// TIA Portal project "SuperSygnalizacjaDomiLechLuka" (V16)

(* hardware
DEVICE "S7-1200 station_2"  S7-1200 Station
   slot 0: "Rack_0"  S7-1200 Rack  Rack  V1.0
   slot 1: "PLC_2"  CPU 1215C AC/DC/Rly  6ES7 215-1BG40-0XB0  V4.4
DEVICE "S7-1200 station_1"  S7-1200 Station
   slot 0: "Rack_0"  S7-1200 Rack  Rack  V1.0
   slot 1: "PLC_1"  CPU 1215C AC/DC/Rly  6ES7 215-1BG40-0XB0  V4.4
*)

// ===== PLC "PLC_1"  CPU 1215C AC/DC/Rly =====

VAR_GLOBAL   // PLC tag table "Default tag table"
   "Clock_Byte" AT %MB0 : Byte;
   "Clock_10Hz" AT %M0.0 : Bool;
   "Clock_5Hz" AT %M0.1 : Bool;
   "Clock_2.5Hz" AT %M0.2 : Bool;
   "Clock_2Hz" AT %M0.3 : Bool;
   "Clock_1.25Hz" AT %M0.4 : Bool;
   "Clock_1Hz" AT %M0.5 : Bool;
   "Clock_0.625Hz" AT %M0.6 : Bool;
   "Clock_0.5Hz" AT %M0.7 : Bool;
   "P3_P4_green" AT %Q0.0 : Bool;
   "P3_P4_red" AT %Q0.1 : Bool;
   "W1_W3_W4_red" AT %Q0.2 : Bool;
   "W1_W3_W4_yellow" AT %Q0.3 : Bool;
   "W1_W3_W4_green" AT %Q0.4 : Bool;
   "W2_W6_red" AT %Q0.5 : Bool;
   "W2_W6_yellow" AT %Q0.6 : Bool;
   "W2_W6_green" AT %Q0.7 : Bool;
   "P2_red" AT %Q1.0 : Bool;
   "Start" AT %M1.0 : Bool;
   "Timer_CV" AT %MD10 : DWord;
   "P2_green" AT %M1.1 : Bool;
   "W7_red" AT %M1.2 : Bool;
   "W7_yellow" AT %M1.3 : Bool;
   "W7_green" AT %M1.4 : Bool;
   "W5_red" AT %M1.5 : Bool;
   "W5_yellow" AT %M1.6 : Bool;
   "W5_green" AT %M1.7 : Bool;
   "P1_red" AT %M2.0 : Bool;
   "P1_green" AT %M2.1 : Bool;
END_VAR

DATA_BLOCK "sent"   // DB1
{ S7_Optimized_Access := 'TRUE' }
VERSION : 0.1
   VAR
      data : Word;
   END_VAR
BEGIN
END_DATA_BLOCK

DATA_BLOCK "recv"   // DB2
{ S7_Optimized_Access := 'TRUE' }
VERSION : 0.1
   VAR
      data : Word;
   END_VAR
BEGIN
END_DATA_BLOCK

// folder: System blocks/Program resources

DATA_BLOCK "IEC_Timer_0_DB"   // DB3
{ S7_Optimized_Access := 'TRUE' }
AUTHOR : Simatic
FAMILY : IEC
NAME : IEC_TMR
VERSION : 1.0
// stored: InstanceOfName IEC_TIMER
"IEC_TIMER"
BEGIN
END_DATA_BLOCK

// folder: (top level)

ORGANIZATION_BLOCK "Main"   // OB1, LAD, ProgramCycle
TITLE = "Main Program Sweep (Cycle)"
{ S7_Optimized_Access := 'TRUE' }
VERSION : 0.1
   VAR_INPUT
      Initial_Call : Bool;   // Initial call of this OB
      Remanence : Bool;   // =True, if remanent data are available
   END_VAR
BEGIN

REGION Network 1: Main timer
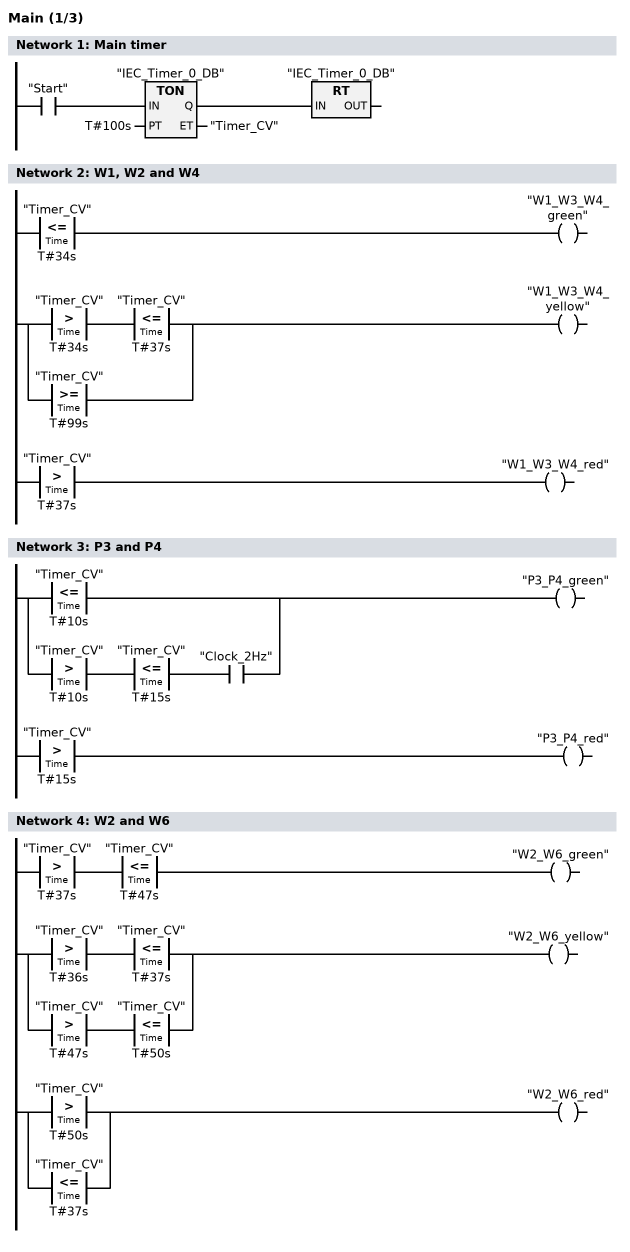
   "IEC_Timer_0_DB".TON(IN := "Start", PT := T#100s, ET => "Timer_CV");
   IF "IEC_Timer_0_DB".Q THEN RESET_TIMER("IEC_Timer_0_DB"); END_IF;
END_REGION

REGION Network 2: W1, W2 and W4
   RUNG wire#powerrail
      { S7_Templates := "SrcType := Time" } LE_Contact(in1 := "Timer_CV", in2 := T#34s)
      Coil( "W1_W3_W4_green" )
   END_RUNG
   RUNG wire#powerrail
      { S7_Templates := "SrcType := Time" } GT_Contact(in1 := "Timer_CV", in2 := T#34s)
      { S7_Templates := "SrcType := Time" } LE_Contact(in1 := "Timer_CV", in2 := T#37s)
      wire#w1
      Coil( "W1_W3_W4_yellow" )
   END_RUNG
   RUNG wire#powerrail
      { S7_Templates := "SrcType := Time" } GE_Contact(in1 := "Timer_CV", in2 := T#99s)
   END_RUNG wire#w1
   RUNG wire#powerrail
      { S7_Templates := "SrcType := Time" } GT_Contact(in1 := "Timer_CV", in2 := T#37s)
      Coil( "W1_W3_W4_red" )
   END_RUNG
   // the same network as SCL:
   "W1_W3_W4_green" := "Timer_CV" <= T#34s;
   "W1_W3_W4_yellow" := (("Timer_CV" > T#34s) AND ("Timer_CV" <= T#37s)) OR ("Timer_CV" >= T#99s);
   "W1_W3_W4_red" := "Timer_CV" > T#37s;
END_REGION

REGION Network 3: P3 and P4
   RUNG wire#powerrail
      { S7_Templates := "SrcType := Time" } LE_Contact(in1 := "Timer_CV", in2 := T#10s)
      wire#w1
      Coil( "P3_P4_green" )
   END_RUNG
   RUNG wire#powerrail
      { S7_Templates := "SrcType := Time" } GT_Contact(in1 := "Timer_CV", in2 := T#10s)
      { S7_Templates := "SrcType := Time" } LE_Contact(in1 := "Timer_CV", in2 := T#15s)
      Contact( "Clock_2Hz" )
   END_RUNG wire#w1
   RUNG wire#powerrail
      { S7_Templates := "SrcType := Time" } GT_Contact(in1 := "Timer_CV", in2 := T#15s)
      Coil( "P3_P4_red" )
   END_RUNG
   // the same network as SCL:
   "P3_P4_green" := ("Timer_CV" <= T#10s) OR (("Timer_CV" > T#10s) AND ("Timer_CV" <= T#15s) AND "Clock_2Hz");
   "P3_P4_red" := "Timer_CV" > T#15s;
END_REGION

REGION Network 4: W2 and W6
   RUNG wire#powerrail
      { S7_Templates := "SrcType := Time" } GT_Contact(in1 := "Timer_CV", in2 := T#37s)
      { S7_Templates := "SrcType := Time" } LE_Contact(in1 := "Timer_CV", in2 := T#47s)
      Coil( "W2_W6_green" )
   END_RUNG
   RUNG wire#powerrail
      { S7_Templates := "SrcType := Time" } GT_Contact(in1 := "Timer_CV", in2 := T#36s)
      { S7_Templates := "SrcType := Time" } LE_Contact(in1 := "Timer_CV", in2 := T#37s)
      wire#w1
      Coil( "W2_W6_yellow" )
   END_RUNG
   RUNG wire#powerrail
      { S7_Templates := "SrcType := Time" } GT_Contact(in1 := "Timer_CV", in2 := T#47s)
      { S7_Templates := "SrcType := Time" } LE_Contact(in1 := "Timer_CV", in2 := T#50s)
   END_RUNG wire#w1
   RUNG wire#powerrail
      { S7_Templates := "SrcType := Time" } GT_Contact(in1 := "Timer_CV", in2 := T#50s)
      wire#w2
      Coil( "W2_W6_red" )
   END_RUNG
   RUNG wire#powerrail
      { S7_Templates := "SrcType := Time" } LE_Contact(in1 := "Timer_CV", in2 := T#37s)
   END_RUNG wire#w2
   // the same network as SCL:
   "W2_W6_green" := ("Timer_CV" > T#37s) AND ("Timer_CV" <= T#47s);
   "W2_W6_yellow" := (("Timer_CV" > T#36s) AND ("Timer_CV" <= T#37s)) OR (("Timer_CV" > T#47s) AND ("Timer_CV" <= T#50s));
   "W2_W6_red" := ("Timer_CV" > T#50s) OR ("Timer_CV" <= T#37s);
END_REGION

REGION Network 5: P2
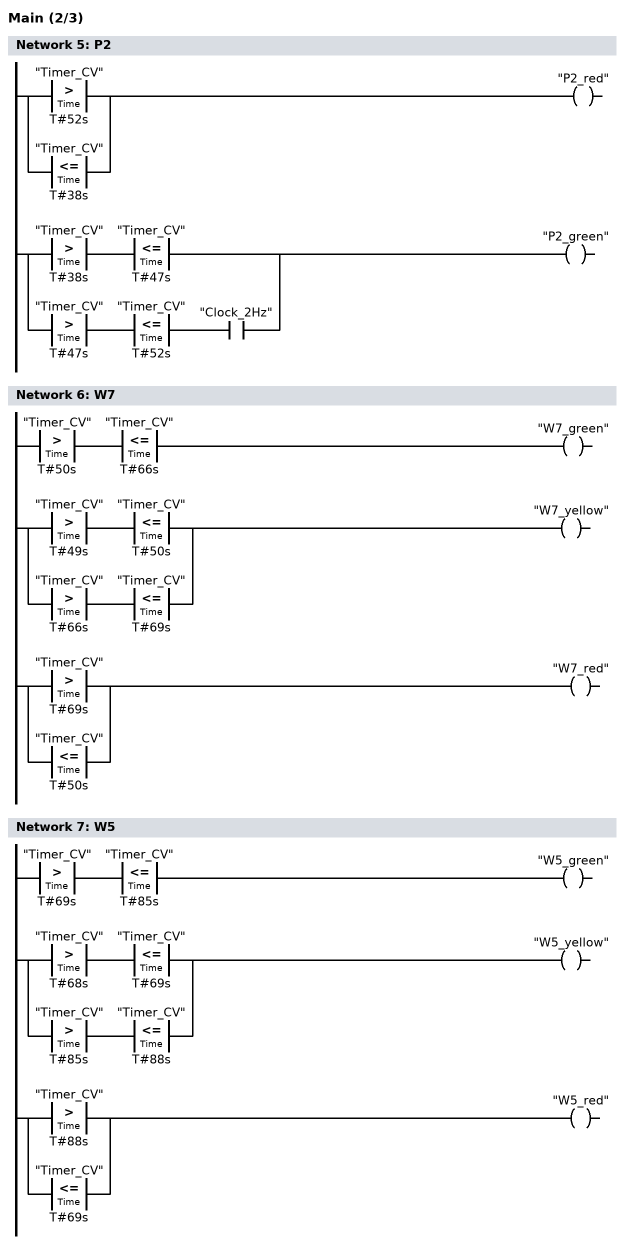
   RUNG wire#powerrail
      { S7_Templates := "SrcType := Time" } GT_Contact(in1 := "Timer_CV", in2 := T#52s)
      wire#w1
      Coil( "P2_red" )
   END_RUNG
   RUNG wire#powerrail
      { S7_Templates := "SrcType := Time" } LE_Contact(in1 := "Timer_CV", in2 := T#38s)
   END_RUNG wire#w1
   RUNG wire#powerrail
      { S7_Templates := "SrcType := Time" } GT_Contact(in1 := "Timer_CV", in2 := T#38s)
      { S7_Templates := "SrcType := Time" } LE_Contact(in1 := "Timer_CV", in2 := T#47s)
      wire#w2
      Coil( "P2_green" )
   END_RUNG
   RUNG wire#powerrail
      { S7_Templates := "SrcType := Time" } GT_Contact(in1 := "Timer_CV", in2 := T#47s)
      { S7_Templates := "SrcType := Time" } LE_Contact(in1 := "Timer_CV", in2 := T#52s)
      Contact( "Clock_2Hz" )
   END_RUNG wire#w2
   // the same network as SCL:
   "P2_red" := ("Timer_CV" > T#52s) OR ("Timer_CV" <= T#38s);
   "P2_green" := (("Timer_CV" > T#38s) AND ("Timer_CV" <= T#47s)) OR (("Timer_CV" > T#47s) AND ("Timer_CV" <= T#52s) AND "Clock_2Hz");
END_REGION

REGION Network 6: W7
   RUNG wire#powerrail
      { S7_Templates := "SrcType := Time" } GT_Contact(in1 := "Timer_CV", in2 := T#50s)
      { S7_Templates := "SrcType := Time" } LE_Contact(in1 := "Timer_CV", in2 := T#66s)
      Coil( "W7_green" )
   END_RUNG
   RUNG wire#powerrail
      { S7_Templates := "SrcType := Time" } GT_Contact(in1 := "Timer_CV", in2 := T#49s)
      { S7_Templates := "SrcType := Time" } LE_Contact(in1 := "Timer_CV", in2 := T#50s)
      wire#w1
      Coil( "W7_yellow" )
   END_RUNG
   RUNG wire#powerrail
      { S7_Templates := "SrcType := Time" } GT_Contact(in1 := "Timer_CV", in2 := T#66s)
      { S7_Templates := "SrcType := Time" } LE_Contact(in1 := "Timer_CV", in2 := T#69s)
   END_RUNG wire#w1
   RUNG wire#powerrail
      { S7_Templates := "SrcType := Time" } GT_Contact(in1 := "Timer_CV", in2 := T#69s)
      wire#w2
      Coil( "W7_red" )
   END_RUNG
   RUNG wire#powerrail
      { S7_Templates := "SrcType := Time" } LE_Contact(in1 := "Timer_CV", in2 := T#50s)
   END_RUNG wire#w2
   // the same network as SCL:
   "W7_green" := ("Timer_CV" > T#50s) AND ("Timer_CV" <= T#66s);
   "W7_yellow" := (("Timer_CV" > T#49s) AND ("Timer_CV" <= T#50s)) OR (("Timer_CV" > T#66s) AND ("Timer_CV" <= T#69s));
   "W7_red" := ("Timer_CV" > T#69s) OR ("Timer_CV" <= T#50s);
END_REGION

REGION Network 7: W5
   RUNG wire#powerrail
      { S7_Templates := "SrcType := Time" } GT_Contact(in1 := "Timer_CV", in2 := T#69s)
      { S7_Templates := "SrcType := Time" } LE_Contact(in1 := "Timer_CV", in2 := T#85s)
      Coil( "W5_green" )
   END_RUNG
   RUNG wire#powerrail
      { S7_Templates := "SrcType := Time" } GT_Contact(in1 := "Timer_CV", in2 := T#68s)
      { S7_Templates := "SrcType := Time" } LE_Contact(in1 := "Timer_CV", in2 := T#69s)
      wire#w1
      Coil( "W5_yellow" )
   END_RUNG
   RUNG wire#powerrail
      { S7_Templates := "SrcType := Time" } GT_Contact(in1 := "Timer_CV", in2 := T#85s)
      { S7_Templates := "SrcType := Time" } LE_Contact(in1 := "Timer_CV", in2 := T#88s)
   END_RUNG wire#w1
   RUNG wire#powerrail
      { S7_Templates := "SrcType := Time" } GT_Contact(in1 := "Timer_CV", in2 := T#88s)
      wire#w2
      Coil( "W5_red" )
   END_RUNG
   RUNG wire#powerrail
      { S7_Templates := "SrcType := Time" } LE_Contact(in1 := "Timer_CV", in2 := T#69s)
   END_RUNG wire#w2
   // the same network as SCL:
   "W5_green" := ("Timer_CV" > T#69s) AND ("Timer_CV" <= T#85s);
   "W5_yellow" := (("Timer_CV" > T#68s) AND ("Timer_CV" <= T#69s)) OR (("Timer_CV" > T#85s) AND ("Timer_CV" <= T#88s));
   "W5_red" := ("Timer_CV" > T#88s) OR ("Timer_CV" <= T#69s);
END_REGION

REGION Network 8: P1
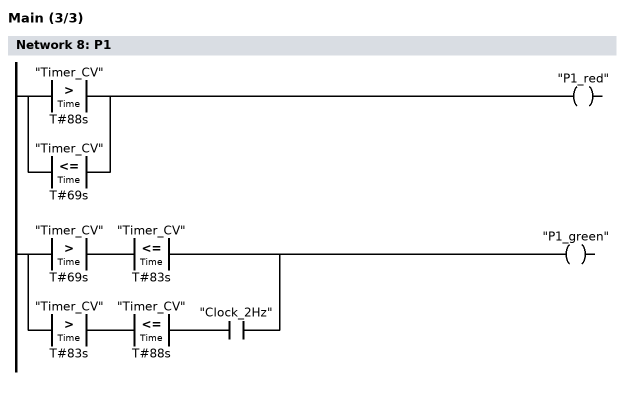
   RUNG wire#powerrail
      { S7_Templates := "SrcType := Time" } GT_Contact(in1 := "Timer_CV", in2 := T#88s)
      wire#w1
      Coil( "P1_red" )
   END_RUNG
   RUNG wire#powerrail
      { S7_Templates := "SrcType := Time" } LE_Contact(in1 := "Timer_CV", in2 := T#69s)
   END_RUNG wire#w1
   RUNG wire#powerrail
      { S7_Templates := "SrcType := Time" } GT_Contact(in1 := "Timer_CV", in2 := T#69s)
      { S7_Templates := "SrcType := Time" } LE_Contact(in1 := "Timer_CV", in2 := T#83s)
      wire#w2
      Coil( "P1_green" )
   END_RUNG
   RUNG wire#powerrail
      { S7_Templates := "SrcType := Time" } GT_Contact(in1 := "Timer_CV", in2 := T#83s)
      { S7_Templates := "SrcType := Time" } LE_Contact(in1 := "Timer_CV", in2 := T#88s)
      Contact( "Clock_2Hz" )
   END_RUNG wire#w2
   // the same network as SCL:
   "P1_red" := ("Timer_CV" > T#88s) OR ("Timer_CV" <= T#69s);
   "P1_green" := (("Timer_CV" > T#69s) AND ("Timer_CV" <= T#83s)) OR (("Timer_CV" > T#83s) AND ("Timer_CV" <= T#88s) AND "Clock_2Hz");
END_REGION
END_ORGANIZATION_BLOCK

// ===== PLC "PLC_2"  CPU 1215C AC/DC/Rly =====

VAR_GLOBAL   // PLC tag table "Default tag table"
   "Clock_Byte" AT %MB0 : Byte;
   "Clock_10Hz" AT %M0.0 : Bool;
   "Clock_5Hz" AT %M0.1 : Bool;
   "Clock_2.5Hz" AT %M0.2 : Bool;
   "Clock_2Hz" AT %M0.3 : Bool;
   "Clock_1.25Hz" AT %M0.4 : Bool;
   "Clock_1Hz" AT %M0.5 : Bool;
   "Clock_0.625Hz" AT %M0.6 : Bool;
   "Clock_0.5Hz" AT %M0.7 : Bool;
END_VAR

DATA_BLOCK "sent"   // DB1
{ S7_Optimized_Access := 'TRUE' }
VERSION : 0.1
   VAR
      data : Word;
   END_VAR
BEGIN
END_DATA_BLOCK

DATA_BLOCK "recv"   // DB2
{ S7_Optimized_Access := 'TRUE' }
VERSION : 0.1
   VAR
      data : Word;
   END_VAR
BEGIN
END_DATA_BLOCK

ORGANIZATION_BLOCK "Main"   // OB1, LAD, ProgramCycle
TITLE = "Main Program Sweep (Cycle)"
{ S7_Optimized_Access := 'TRUE' }
VERSION : 0.1
   VAR_INPUT
      Initial_Call : Bool;   // Initial call of this OB
      Remanence : Bool;   // =True, if remanent data are available
   END_VAR
BEGIN
END_ORGANIZATION_BLOCK